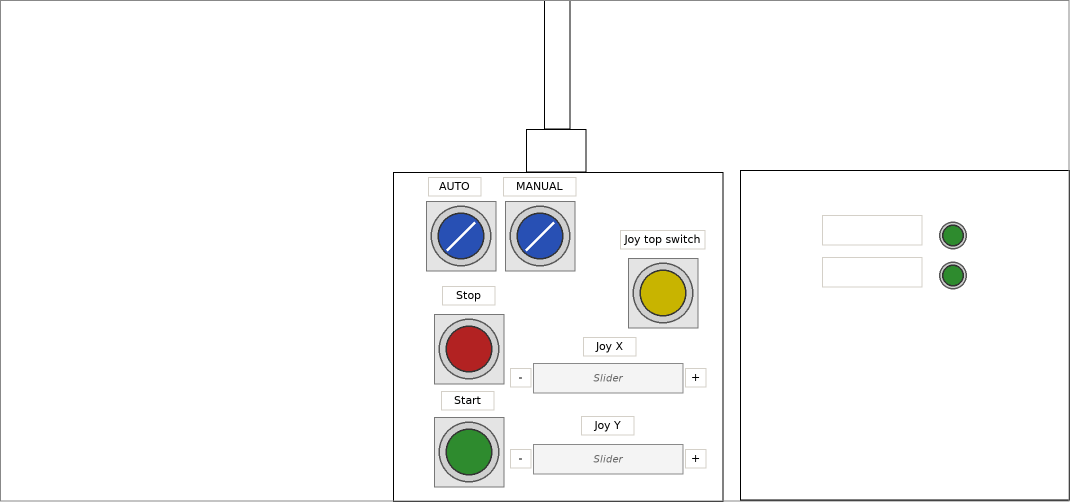
VISUALIZATION Visualization  // 1070x502
    RoundedRectangle (393,172 330x330)
    RotarySwitch (426,201 70x70), variable: G_Task_1.bAuto, behaviour: TOGGLE, style: Switch-RotarySwitch-Blue
    PushSwitch (434,417 70x70), variable: G_Task_1.bStart, behaviour: TOGGLE, style: Switch-PushSwitch-Green
    PushSwitch (434,314 70x70), variable: G_Task_1.bStop, behaviour: TOGGLE, style: Switch-PushSwitch-Red
    RotarySwitch (505,201 70x70), variable: G_Task_1.bManual, behaviour: TOGGLE, style: Switch-RotarySwitch-Blue
    Slider (533,444 150x30), variable: G_Task_1.fJoyY, input disabled if: G_Task_1.bJoyNotActive, scale -1..1
    Slider (533,363 150x30), variable: G_Task_1.fJoyX, input disabled if: G_Task_1.bJoyNotActive, scale -1..1
    Rectangle (526,129 60x43)
    Rectangle (544,0 26x129)
    Textfield (442,286 53x19), "Stop"
    Textfield (441,391 53x19), "Start"
    Textfield (583,337 53x19), "Joy X"
    Textfield (581,416 53x19), "Joy Y"
    PushSwitchLed (628,258 70x70), variable: G_Task_1.bJoyActive, behaviour: TOGGLE, style: Switch-PushSwitchLed-Yellow
    Textfield (620,230 85x19), "Joy top switch"
    Textfield (685,368 21x19), "+"
    Textfield (685,449 21x19), "+"
    Textfield (510,449 21x19), "-"
    Textfield (510,368 21x19), "-"
    Textfield (428,177 53x19), "AUTO"
    Textfield (503,177 73x19), "MANUAL"
    RoundedRectangle (740,170 330x330)
    Label (756,214 63x30), "Mode:"
    Label (738,253 90x38), "Status:"
    Textfield (822,215 100x30)
    Lamp1 (937,215 32x41), style: Lamp-Lamp1-Green
    Textfield (822,257 100x30)
    Lamp1 (937,255 32x41), style: Lamp-Lamp1-Green
END_VISUALIZATION

(* stored: Version 1.1.0.1, ProductVersion 3.1.4024.12
   Visu Visualization: Id {81918428-894a-4d31-8869-aaee674000f5} *)
